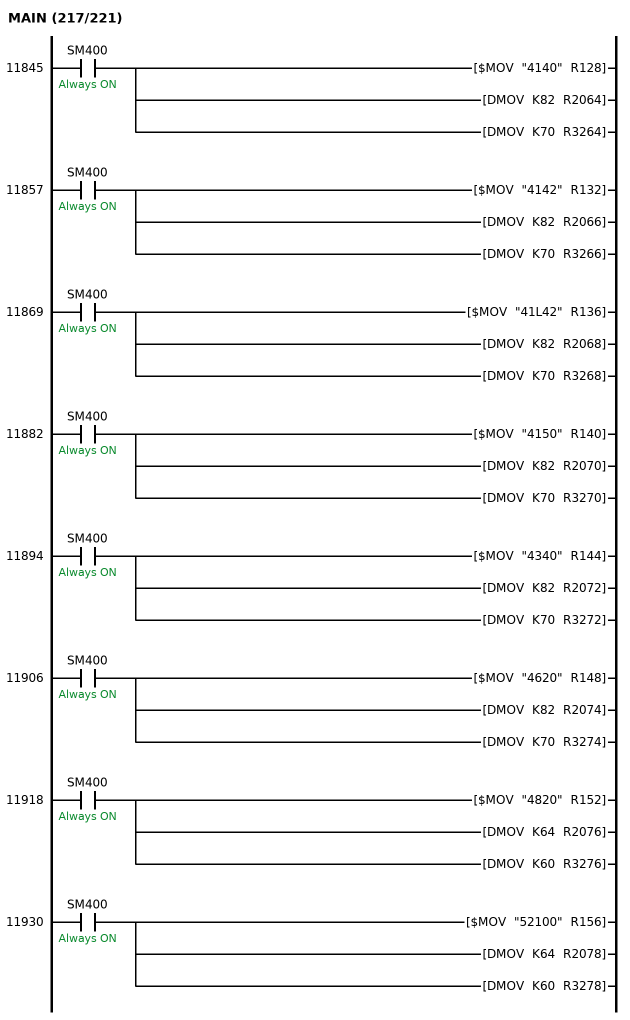
[picture p216: ladder of MAIN, rungs at steps 11845 to 11930]
11845 LD      SM400  ; Always ON
      $MOV    "4140" R128
      DMOV    K82 R2064
      DMOV    K70 R3264
11857 LD      SM400  ; Always ON
      $MOV    "4142" R132
      DMOV    K82 R2066
      DMOV    K70 R3266
11869 LD      SM400  ; Always ON
      $MOV    "41L42" R136
      DMOV    K82 R2068
      DMOV    K70 R3268
11882 LD      SM400  ; Always ON
      $MOV    "4150" R140
      DMOV    K82 R2070
      DMOV    K70 R3270
11894 LD      SM400  ; Always ON
      $MOV    "4340" R144
      DMOV    K82 R2072
      DMOV    K70 R3272
11906 LD      SM400  ; Always ON
      $MOV    "4620" R148
      DMOV    K82 R2074
      DMOV    K70 R3274
11918 LD      SM400  ; Always ON
      $MOV    "4820" R152
      DMOV    K64 R2076
      DMOV    K60 R3276
11930 LD      SM400  ; Always ON
      $MOV    "52100" R156
      DMOV    K64 R2078
      DMOV    K60 R3278
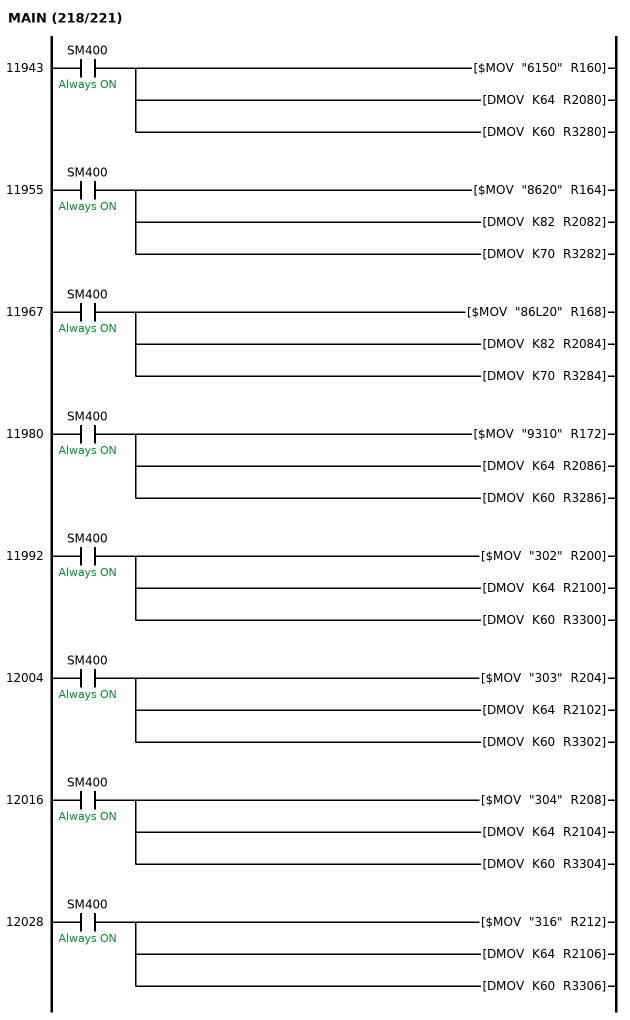
11943 LD      SM400  ; Always ON
      $MOV    "6150" R160
      DMOV    K64 R2080
      DMOV    K60 R3280
11955 LD      SM400  ; Always ON
      $MOV    "8620" R164
      DMOV    K82 R2082
      DMOV    K70 R3282
11967 LD      SM400  ; Always ON
      $MOV    "86L20" R168
      DMOV    K82 R2084
      DMOV    K70 R3284
11980 LD      SM400  ; Always ON
      $MOV    "9310" R172
      DMOV    K64 R2086
      DMOV    K60 R3286
11992 LD      SM400  ; Always ON
      $MOV    "302" R200
      DMOV    K64 R2100
      DMOV    K60 R3300
12004 LD      SM400  ; Always ON
      $MOV    "303" R204
      DMOV    K64 R2102
      DMOV    K60 R3302
12016 LD      SM400  ; Always ON
      $MOV    "304" R208
      DMOV    K64 R2104
      DMOV    K60 R3304
12028 LD      SM400  ; Always ON
      $MOV    "316" R212
      DMOV    K64 R2106
      DMOV    K60 R3306
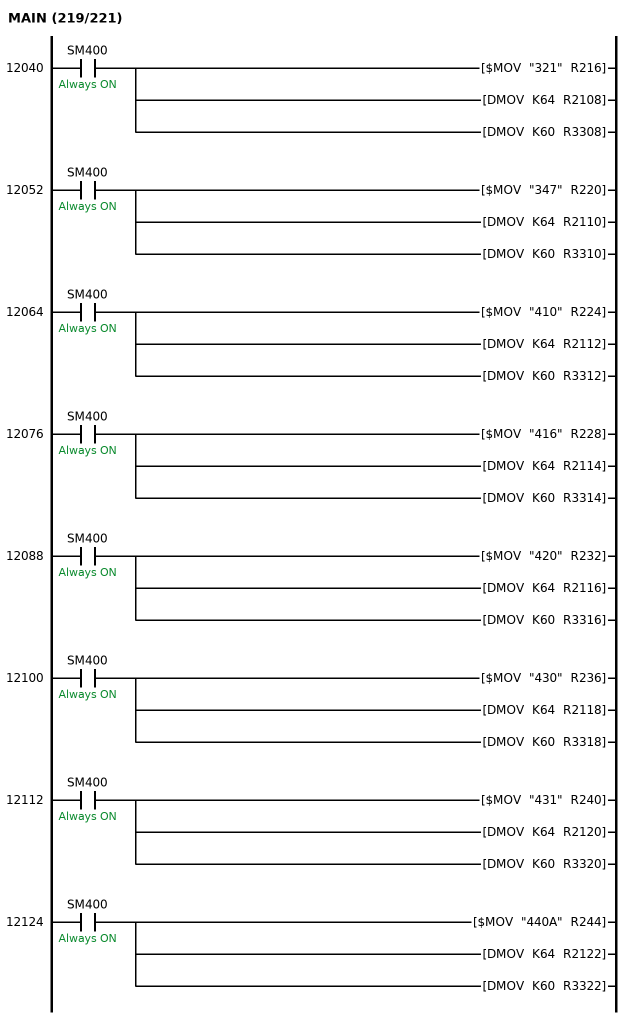
12040 LD      SM400  ; Always ON
      $MOV    "321" R216
      DMOV    K64 R2108
      DMOV    K60 R3308
12052 LD      SM400  ; Always ON
      $MOV    "347" R220
      DMOV    K64 R2110
      DMOV    K60 R3310
12064 LD      SM400  ; Always ON
      $MOV    "410" R224
      DMOV    K64 R2112
      DMOV    K60 R3312
12076 LD      SM400  ; Always ON
      $MOV    "416" R228
      DMOV    K64 R2114
      DMOV    K60 R3314
12088 LD      SM400  ; Always ON
      $MOV    "420" R232
      DMOV    K64 R2116
      DMOV    K60 R3316
12100 LD      SM400  ; Always ON
      $MOV    "430" R236
      DMOV    K64 R2118
      DMOV    K60 R3318
12112 LD      SM400  ; Always ON
      $MOV    "431" R240
      DMOV    K64 R2120
      DMOV    K60 R3320
12124 LD      SM400  ; Always ON
      $MOV    "440A" R244
      DMOV    K64 R2122
      DMOV    K60 R3322
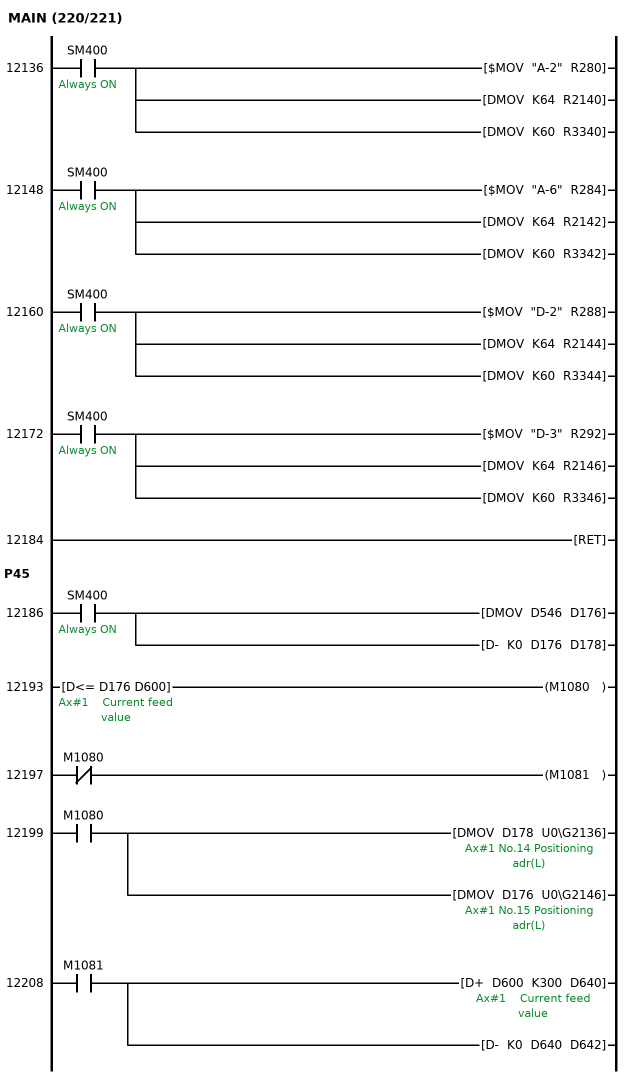
12136 LD      SM400  ; Always ON
      $MOV    "A-2" R280
      DMOV    K64 R2140
      DMOV    K60 R3340
12148 LD      SM400  ; Always ON
      $MOV    "A-6" R284
      DMOV    K64 R2142
      DMOV    K60 R3342
12160 LD      SM400  ; Always ON
      $MOV    "D-2" R288
      DMOV    K64 R2144
      DMOV    K60 R3344
12172 LD      SM400  ; Always ON
      $MOV    "D-3" R292
      DMOV    K64 R2146
      DMOV    K60 R3346
12184 RET
      P45
12186 LD      SM400  ; Always ON
      DMOV    D546 D176
      D-      K0 D176 D178
12193 LDD<=   D176 D600  ; Ax#1    Current feed    value
      OUT     M1080
12197 LDI     M1080
      OUT     M1081
12199 LD      M1080
      DMOV    D178 U0\G2136  ; Ax#1 No.14 Positioning adr(L)
      DMOV    D176 U0\G2146  ; Ax#1 No.15 Positioning adr(L)
12208 LD      M1081
      D+      D600 K300 D640
      D-      K0 D640 D642
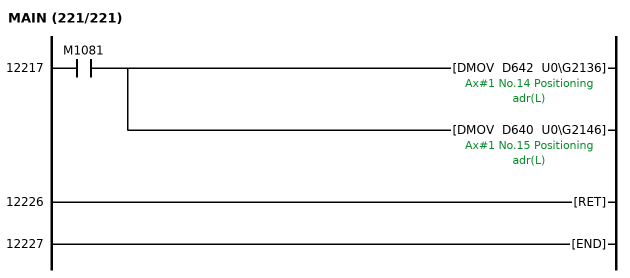
12217 LD      M1081
      DMOV    D642 U0\G2136
      DMOV    D640 U0\G2146
12226 RET
12227 END
END_PROGRAM

PROGRAM HMS
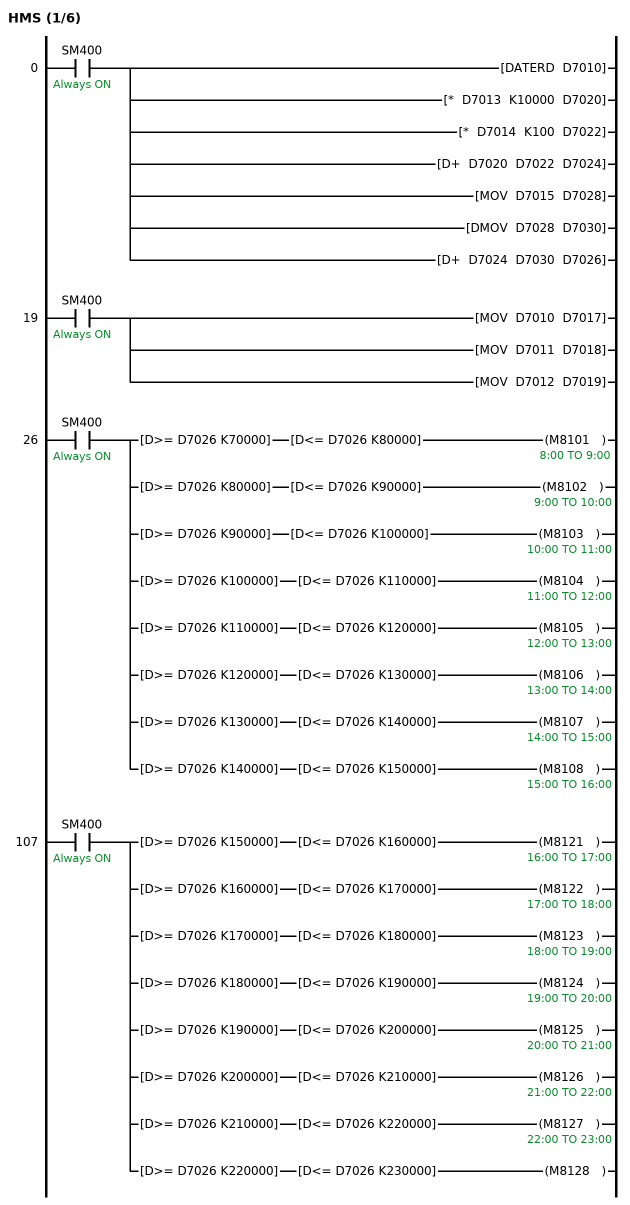
0     LD      SM400  ; Always ON
      DATERD  D7010
      *       D7013 K10000 D7020
      *       D7014 K100 D7022
      D+      D7020 D7022 D7024
      MOV     D7015 D7028
      DMOV    D7028 D7030
      D+      D7024 D7030 D7026
19    LD      SM400  ; Always ON
      MOV     D7010 D7017
      MOV     D7011 D7018
      MOV     D7012 D7019
26    LD      SM400  ; Always ON
      MPS
      ANDD>=  D7026 K70000
      ANDD<=  D7026 K80000
      OUT     M8101  ; 8:00 TO 9:00
      MRD
      ANDD>=  D7026 K80000
      ANDD<=  D7026 K90000
      OUT     M8102  ; 9:00 TO 10:00
      MRD
      ANDD>=  D7026 K90000
      ANDD<=  D7026 K100000
      OUT     M8103  ; 10:00 TO 11:00
      MRD
      ANDD>=  D7026 K100000
      ANDD<=  D7026 K110000
      OUT     M8104  ; 11:00 TO 12:00
      MRD
      ANDD>=  D7026 K110000
      ANDD<=  D7026 K120000
      OUT     M8105  ; 12:00 TO 13:00
      MRD
      ANDD>=  D7026 K120000
      ANDD<=  D7026 K130000
      OUT     M8106  ; 13:00 TO 14:00
      MRD
      ANDD>=  D7026 K130000
      ANDD<=  D7026 K140000
      OUT     M8107  ; 14:00 TO 15:00
      MPP
      ANDD>=  D7026 K140000
      ANDD<=  D7026 K150000
      OUT     M8108  ; 15:00 TO 16:00
107   LD      SM400  ; Always ON
      MPS
      ANDD>=  D7026 K150000
      ANDD<=  D7026 K160000
      OUT     M8121  ; 16:00 TO 17:00
      MRD
      ANDD>=  D7026 K160000
      ANDD<=  D7026 K170000
      OUT     M8122  ; 17:00 TO 18:00
      MRD
      ANDD>=  D7026 K170000
      ANDD<=  D7026 K180000
      OUT     M8123  ; 18:00 TO 19:00
      MRD
      ANDD>=  D7026 K180000
      ANDD<=  D7026 K190000
      OUT     M8124  ; 19:00 TO 20:00
      MRD
      ANDD>=  D7026 K190000
      ANDD<=  D7026 K200000
      OUT     M8125  ; 20:00 TO 21:00
      MRD
      ANDD>=  D7026 K200000
      ANDD<=  D7026 K210000
      OUT     M8126  ; 21:00 TO 22:00
      MRD
      ANDD>=  D7026 K210000
      ANDD<=  D7026 K220000
      OUT     M8127  ; 22:00 TO 23:00
      MPP
      ANDD>=  D7026 K220000
      ANDD<=  D7026 K230000
      OUT     M8128
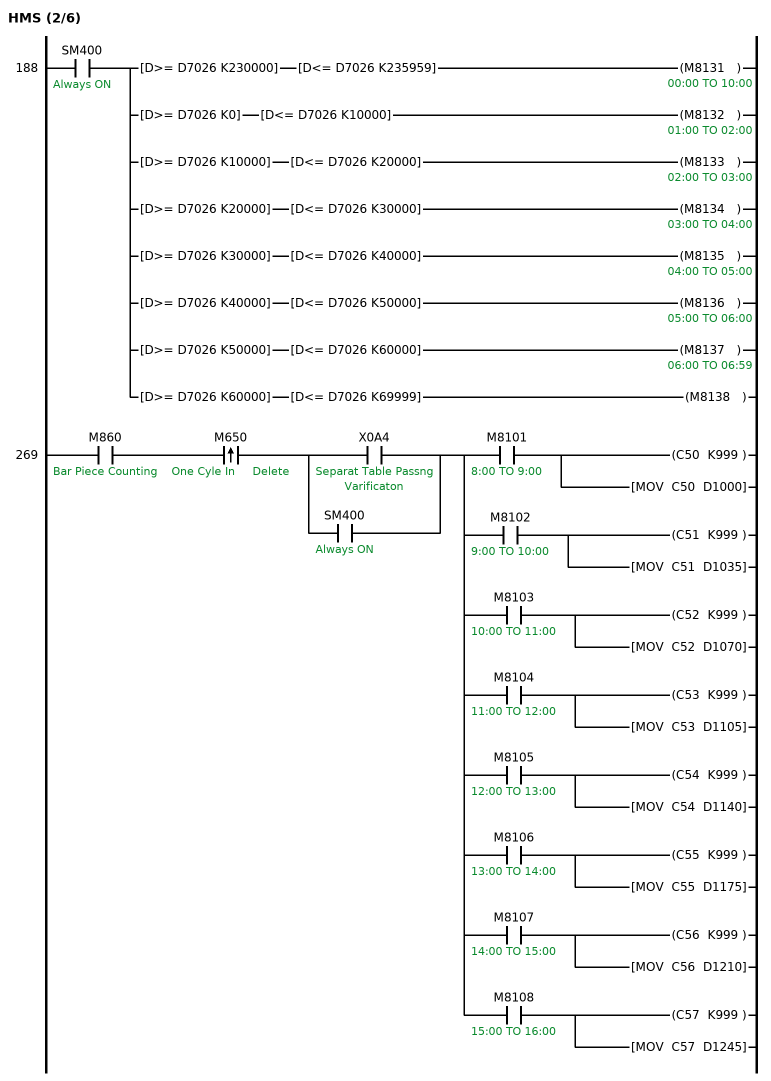
188   LD      SM400  ; Always ON
      MPS
      ANDD>=  D7026 K230000
      ANDD<=  D7026 K235959
      OUT     M8131  ; 00:00 TO 10:00
      MRD
      ANDD>=  D7026 K0
      ANDD<=  D7026 K10000
      OUT     M8132  ; 01:00 TO 02:00
      MRD
      ANDD>=  D7026 K10000
      ANDD<=  D7026 K20000
      OUT     M8133  ; 02:00 TO 03:00
      MRD
      ANDD>=  D7026 K20000
      ANDD<=  D7026 K30000
      OUT     M8134  ; 03:00 TO 04:00
      MRD
      ANDD>=  D7026 K30000
      ANDD<=  D7026 K40000
      OUT     M8135  ; 04:00 TO 05:00
      MRD
      ANDD>=  D7026 K40000
      ANDD<=  D7026 K50000
      OUT     M8136  ; 05:00 TO 06:00
      MRD
      ANDD>=  D7026 K50000
      ANDD<=  D7026 K60000
      OUT     M8137  ; 06:00 TO 06:59
      MPP
      ANDD>=  D7026 K60000
      ANDD<=  D7026 K69999
      OUT     M8138
269   LD      M860  ; Bar Piece Counting
      ANDP    M650  ; One Cyle In     Delete
      LD      X0A4  ; Separat Table Passng Varificaton
      OR      SM400  ; Always ON
      ANB
      MPS
      AND     M8101  ; 8:00 TO 9:00
      OUT     C50 K999
      MOV     C50 D1000
      MRD
      AND     M8102  ; 9:00 TO 10:00
      OUT     C51 K999
      MOV     C51 D1035
      MRD
      AND     M8103  ; 10:00 TO 11:00
      OUT     C52 K999
      MOV     C52 D1070
      MRD
      AND     M8104  ; 11:00 TO 12:00
      OUT     C53 K999
      MOV     C53 D1105
      MRD
      AND     M8105  ; 12:00 TO 13:00
      OUT     C54 K999
      MOV     C54 D1140
      MRD
      AND     M8106  ; 13:00 TO 14:00
      OUT     C55 K999
      MOV     C55 D1175
      MRD
      AND     M8107  ; 14:00 TO 15:00
      OUT     C56 K999
      MOV     C56 D1210
      MPP
      AND     M8108  ; 15:00 TO 16:00
      OUT     C57 K999
      MOV     C57 D1245
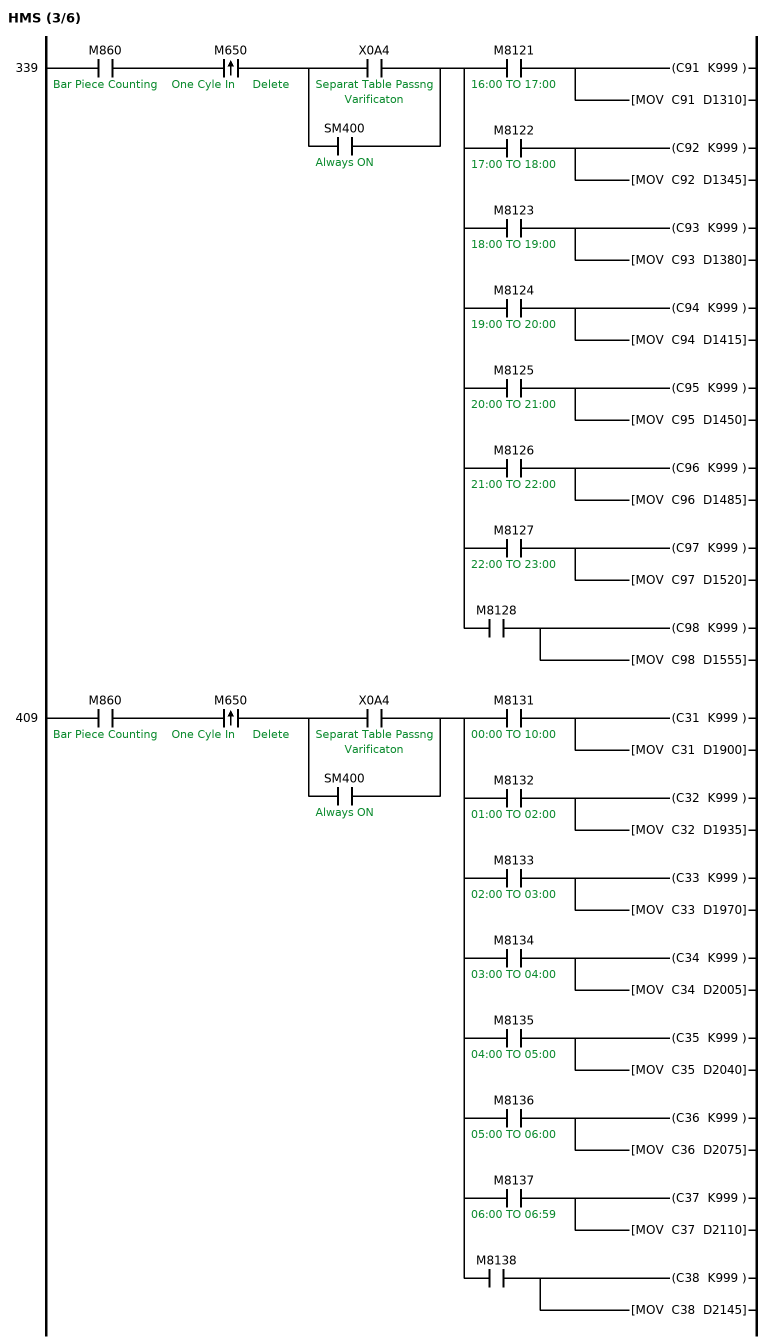
339   LD      M860  ; Bar Piece Counting
      ANDP    M650  ; One Cyle In     Delete
      LD      X0A4  ; Separat Table Passng Varificaton
      OR      SM400  ; Always ON
      ANB
      MPS
      AND     M8121  ; 16:00 TO 17:00
      OUT     C91 K999
      MOV     C91 D1310
      MRD
      AND     M8122  ; 17:00 TO 18:00
      OUT     C92 K999
      MOV     C92 D1345
      MRD
      AND     M8123  ; 18:00 TO 19:00
      OUT     C93 K999
      MOV     C93 D1380
      MRD
      AND     M8124  ; 19:00 TO 20:00
      OUT     C94 K999
      MOV     C94 D1415
      MRD
      AND     M8125  ; 20:00 TO 21:00
      OUT     C95 K999
      MOV     C95 D1450
      MRD
      AND     M8126  ; 21:00 TO 22:00
      OUT     C96 K999
      MOV     C96 D1485
      MRD
      AND     M8127  ; 22:00 TO 23:00
      OUT     C97 K999
      MOV     C97 D1520
      MPP
      AND     M8128
      OUT     C98 K999
      MOV     C98 D1555
409   LD      M860  ; Bar Piece Counting
      ANDP    M650  ; One Cyle In     Delete
      LD      X0A4  ; Separat Table Passng Varificaton
      OR      SM400  ; Always ON
      ANB
      MPS
      AND     M8131  ; 00:00 TO 10:00
      OUT     C31 K999
      MOV     C31 D1900
      MRD
      AND     M8132  ; 01:00 TO 02:00
      OUT     C32 K999
      MOV     C32 D1935
      MRD
      AND     M8133  ; 02:00 TO 03:00
      OUT     C33 K999
      MOV     C33 D1970
      MRD
      AND     M8134  ; 03:00 TO 04:00
      OUT     C34 K999
      MOV     C34 D2005
      MRD
      AND     M8135  ; 04:00 TO 05:00
      OUT     C35 K999
      MOV     C35 D2040
      MRD
      AND     M8136  ; 05:00 TO 06:00
      OUT     C36 K999
      MOV     C36 D2075
      MRD
      AND     M8137  ; 06:00 TO 06:59
      OUT     C37 K999
      MOV     C37 D2110
      MPP
      AND     M8138
      OUT     C38 K999
      MOV     C38 D2145
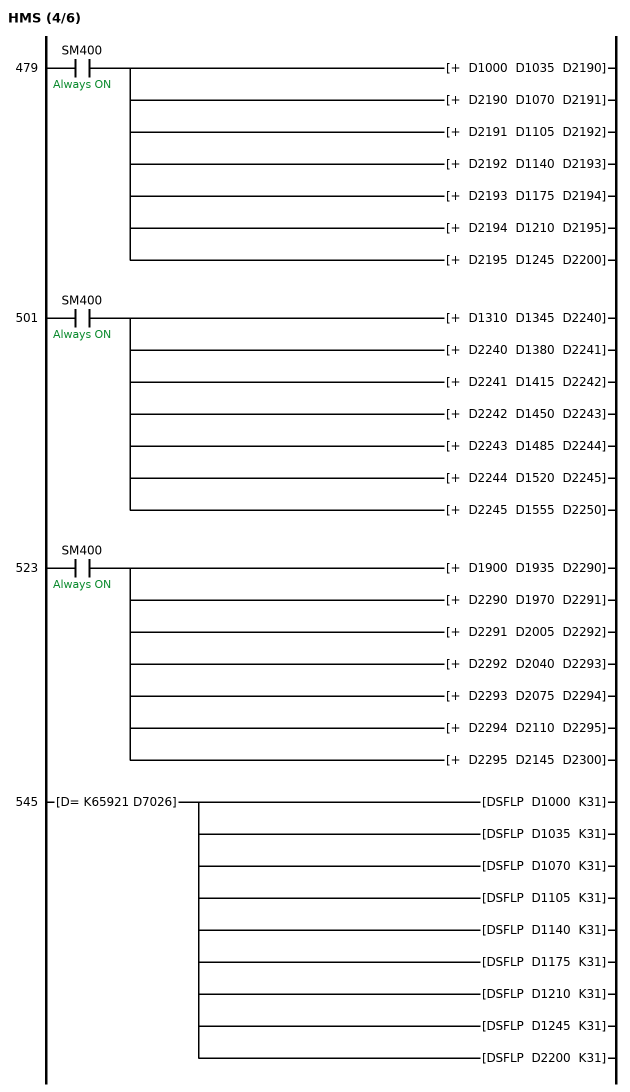
479   LD      SM400  ; Always ON
      +       D1000 D1035 D2190
      +       D2190 D1070 D2191
      +       D2191 D1105 D2192
      +       D2192 D1140 D2193
      +       D2193 D1175 D2194
      +       D2194 D1210 D2195
      +       D2195 D1245 D2200
501   LD      SM400  ; Always ON
      +       D1310 D1345 D2240
      +       D2240 D1380 D2241
      +       D2241 D1415 D2242
      +       D2242 D1450 D2243
      +       D2243 D1485 D2244
      +       D2244 D1520 D2245
      +       D2245 D1555 D2250
523   LD      SM400  ; Always ON
      +       D1900 D1935 D2290
      +       D2290 D1970 D2291
      +       D2291 D2005 D2292
      +       D2292 D2040 D2293
      +       D2293 D2075 D2294
      +       D2294 D2110 D2295
      +       D2295 D2145 D2300
545   LDD=    K65921 D7026
      DSFLP   D1000 K31
      DSFLP   D1035 K31
      DSFLP   D1070 K31
      DSFLP   D1105 K31
      DSFLP   D1140 K31
      DSFLP   D1175 K31
      DSFLP   D1210 K31
      DSFLP   D1245 K31
      DSFLP   D2200 K31
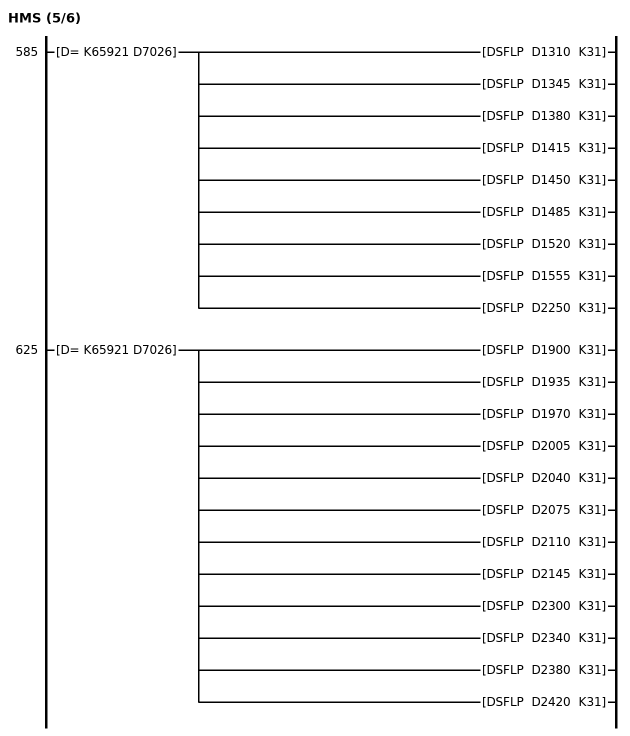
585   LDD=    K65921 D7026
      DSFLP   D1310 K31
      DSFLP   D1345 K31
      DSFLP   D1380 K31
      DSFLP   D1415 K31
      DSFLP   D1450 K31
      DSFLP   D1485 K31
      DSFLP   D1520 K31
      DSFLP   D1555 K31
      DSFLP   D2250 K31
625   LDD=    K65921 D7026
      DSFLP   D1900 K31
      DSFLP   D1935 K31
      DSFLP   D1970 K31
      DSFLP   D2005 K31
      DSFLP   D2040 K31
      DSFLP   D2075 K31
      DSFLP   D2110 K31
      DSFLP   D2145 K31
      DSFLP   D2300 K31
      DSFLP   D2340 K31
      DSFLP   D2380 K31
      DSFLP   D2420 K31
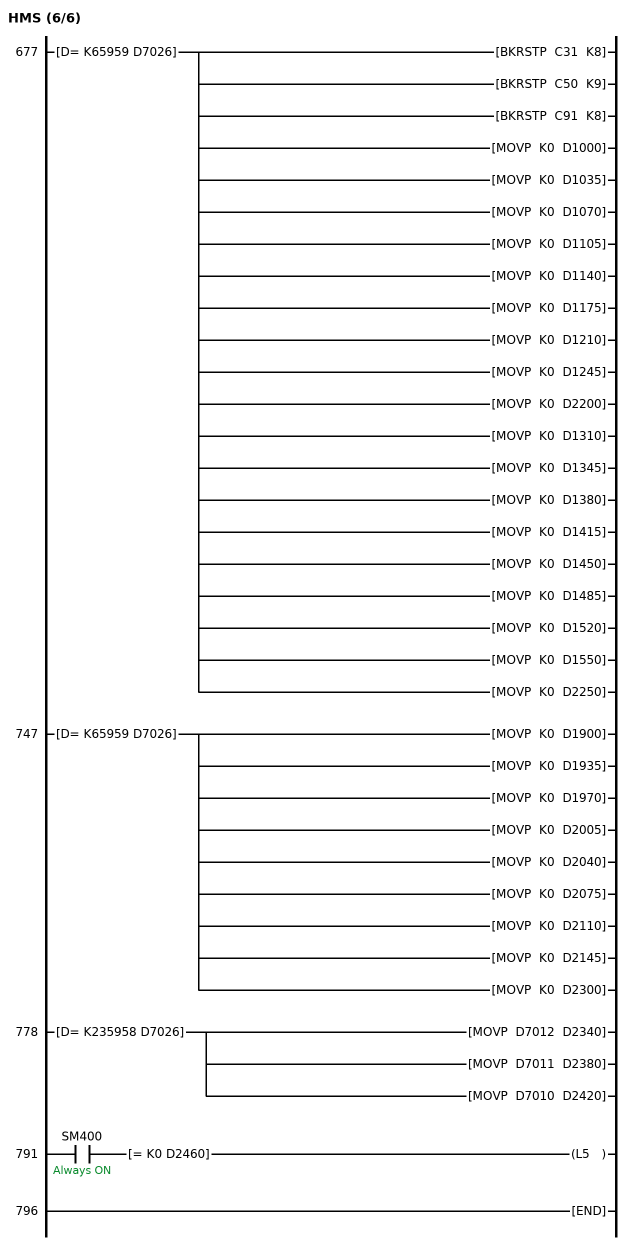
677   LDD=    K65959 D7026
      BKRSTP  C31 K8
      BKRSTP  C50 K9
      BKRSTP  C91 K8
      MOVP    K0 D1000
      MOVP    K0 D1035
      MOVP    K0 D1070
      MOVP    K0 D1105
      MOVP    K0 D1140
      MOVP    K0 D1175
      MOVP    K0 D1210
      MOVP    K0 D1245
      MOVP    K0 D2200
      MOVP    K0 D1310
      MOVP    K0 D1345
      MOVP    K0 D1380
      MOVP    K0 D1415
      MOVP    K0 D1450
      MOVP    K0 D1485
      MOVP    K0 D1520
      MOVP    K0 D1550
      MOVP    K0 D2250
747   LDD=    K65959 D7026
      MOVP    K0 D1900
      MOVP    K0 D1935
      MOVP    K0 D1970
      MOVP    K0 D2005
      MOVP    K0 D2040
      MOVP    K0 D2075
      MOVP    K0 D2110
      MOVP    K0 D2145
      MOVP    K0 D2300
778   LDD=    K235958 D7026
      MOVP    D7012 D2340
      MOVP    D7011 D2380
      MOVP    D7010 D2420
791   LD      SM400  ; Always ON
      AND=    K0 D2460
      OUT     L5
796   END
END_PROGRAM

// device comments not shown above
B201  ; Saw Head Fwd/Bwd  Enable
B202  ; GFC Wise Clamp/Unclamp Enable
B203  ; GFC feed Fwd/Bwd Enable
B204  ; Lader Up/Dn enable
B205  ; Work Stop Fwd/Bwd Enable
B206  ; Float wise On/Off Enable
B207  ; Float work On/Off Enable
B208  ; Seperation Trim/work Enable
B20B  ; Mist ON/Off Enable
B20C  ; Air Blow On/Off Enable
B210  ; Rotary Table fwd/ bwd  Enable
B211  ; Rotary Table ON/ OFF  Enable
B212  ; Lifting Enable
D5100  ; Job ListData    Table
